// TwinCAT 3 PLC project PLC1_AssemblyLine
// Title: PLC1_AssemblyLine
// Company: Beckhoff Automation GmbH & Co. KG
// ProjectVersion: 1.0.0.0
// Description: Sample plc for the TcHmi_AssemblyLine training project
// ProgramVersion: 3.1.4020.10
// libraries:
//   Tc2_MC2, * (Beckhoff Automation GmbH)
//   Tc2_Standard, * (Beckhoff Automation GmbH)
//   Tc2_System, * (Beckhoff Automation GmbH)
//   Tc3_EventLogger, * (Beckhoff Automation GmbH)
//   Tc3_Module, * (Beckhoff Automation GmbH)
// project tree:
//   DUTs/ E_FeederAutoState.TcDUT, E_AxisMode.TcDUT, E_StationState.TcDUT, ST_HmiAxisInfo.TcDUT, ST_HmiFeederInfo.TcDUT, ST_Hmi.TcDUT, ST_HmiAutomaticMode.TcDUT, ST_HmiFeederRecipe.TcDUT, ST_HmiManualMode.TcDUT, ST_HmiOperationMode.TcDUT
//   GVLs/ GVL.TcGVL
//   / PlcTask.TcTTO
//   POUs/ deleteme.TcPOU, FB_Axis.TcPOU, FB_Feeder.TcPOU, MAIN.TcPOU
//   Project Information/ F_GetCompany.TcPOU, F_GetTitle.TcPOU, F_GetVersion.TcPOU
//   Version/ Global_Version.TcGVL
// real-time tasks:
//   TASK PlcTask: cycle T#10ms, priority 8, ADS port 350
// motion (NC):
//   TASK NC-Task-SAF: cycle T#2ms, priority 4, ADS port 501
//   TASK NC-Task-SVB: cycle T#10ms, priority 10, ADS port 511
//   AXIS Feeder1_AxisX (id 1)
//     OtherSettings: AllowMotionCmdToSlave=true
//     encoder EncType=1
//       SoftEndMinControl: Enable=true
//       SoftEndMaxControl: Enable=true, Range=1000
//     drive DrvType=5
//       TimeComp: TaskDelayCycles=1
//     controller CtrType=1
//       CtrPara: PriorControlFactor=1
//         Observer: BandWidth=20
//   AXIS Feeder1_AxisY (id 2)
//     OtherSettings: AllowMotionCmdToSlave=true
//     encoder EncType=1
//       SoftEndMinControl: Enable=true
//       SoftEndMaxControl: Enable=true, Range=1000
//     drive DrvType=5
//       TimeComp: TaskDelayCycles=1
//     controller CtrType=1
//       CtrPara: PriorControlFactor=1
//         Observer: BandWidth=20
//   AXIS Feeder2_AxisX (id 3)
//     OtherSettings: AllowMotionCmdToSlave=true
//     encoder EncType=1
//       SoftEndMinControl: Enable=true
//       SoftEndMaxControl: Enable=true, Range=1000
//     drive DrvType=5
//       TimeComp: TaskDelayCycles=1
//     controller CtrType=1
//       CtrPara: PriorControlFactor=1
//         Observer: BandWidth=20
//   AXIS Feeder2_AxisY (id 4)
//     OtherSettings: AllowMotionCmdToSlave=true
//     encoder EncType=1
//       SoftEndMinControl: Enable=true
//       SoftEndMaxControl: Enable=true, Range=1000
//     drive DrvType=5
//       TimeComp: TaskDelayCycles=1
//     controller CtrType=1
//       CtrPara: PriorControlFactor=1
//         Observer: BandWidth=20
// variable links:
//   PLC1_AssemblyLine/PLC1_AssemblyLine Instance <-> NC-Task-SAF/Axes/Feeder1_AxisX
//     PlcTask Inputs/MAIN.fbFeeders[1].fbAxisX.stAxis.NcToPlc <-> Outputs/ToPlc
//     PlcTask Outputs/MAIN.fbFeeders[1].fbAxisX.stAxis.PlcToNc <-> Inputs/FromPlc
//   PLC1_AssemblyLine/PLC1_AssemblyLine Instance <-> NC-Task-SAF/Axes/Feeder1_AxisY
//     PlcTask Inputs/MAIN.fbFeeders[1].fbAxisY.stAxis.NcToPlc <-> Outputs/ToPlc
//     PlcTask Outputs/MAIN.fbFeeders[1].fbAxisY.stAxis.PlcToNc <-> Inputs/FromPlc
//   PLC1_AssemblyLine/PLC1_AssemblyLine Instance <-> NC-Task-SAF/Axes/Feeder2_AxisX
//     PlcTask Inputs/MAIN.fbFeeders[2].fbAxisX.stAxis.NcToPlc <-> Outputs/ToPlc
//     PlcTask Outputs/MAIN.fbFeeders[2].fbAxisX.stAxis.PlcToNc <-> Inputs/FromPlc
//   PLC1_AssemblyLine/PLC1_AssemblyLine Instance <-> NC-Task-SAF/Axes/Feeder2_AxisY
//     PlcTask Inputs/MAIN.fbFeeders[2].fbAxisY.stAxis.NcToPlc <-> Outputs/ToPlc
//     PlcTask Outputs/MAIN.fbFeeders[2].fbAxisY.stAxis.PlcToNc <-> Inputs/FromPlc

CONFIGURATION PLC1_AssemblyLine
    RESOURCE PLC ON TwinCAT3
        TASK PlcTask(INTERVAL := T#10ms, PRIORITY := 8);
        PROGRAM MAIN WITH PlcTask : MAIN;
    END_RESOURCE
END_CONFIGURATION

// ---- DUTs/E_FeederAutoState.TcDUT
{attribute 'qualified_only'}
TYPE E_FeederAutoState :
(
	eState0_Reset				:= 0,
	eState1_MoveBackToTop		:= 1,
	eState2_MoveToTarget1PosX	:= 2,
	eState3_MoveToTarget1PosY	:= 3,
	eState4_Grab				:= 4,
	eState5_MoveBackToTop		:= 5,
	eState6_MoveToTarget2PosX	:= 6,
	eState7_MoveToTarget2PosY	:= 7,
	eState8_Place				:= 8
);
END_TYPE

// ---- DUTs/E_AxisMode.TcDUT
{attribute 'qualified_only'}
TYPE E_AxisMode :
(
	INIT,
	ENABLE,
	JOG,
	POSITIONING,
	STOP,
	RESET,
	ERROR
);
END_TYPE

// ---- DUTs/E_StationState.TcDUT
{attribute 'qualified_only'}
TYPE E_StationState :
(
	eAuto	:= 0,
	eManual := 1,
	eStop	:= 2	
);
END_TYPE

// ---- DUTs/ST_HmiAxisInfo.TcDUT
TYPE ST_HmiAxisInfo :
STRUCT
	//Actual position
	fActPosition	: LREAL;
	//Actual velocity
	fActVelocity	: LREAL;
	//Current state of axis
	nAxisState		: UDINT;
	//Current mode of axis
	eAxisMode		: E_AxisMode;
END_STRUCT
END_TYPE

// ---- DUTs/ST_HmiFeederInfo.TcDUT
TYPE ST_HmiFeederInfo :
STRUCT
	//Bundled information about axis X
	stAxisX				: ST_HmiAxisInfo;
	
	//Bundled information about axis Y
	stAxisY				: ST_HmiAxisInfo;
	
	//Information about the gripper
	bGripperIsClosed	: BOOL;
END_STRUCT
END_TYPE

// ---- DUTs/ST_Hmi.TcDUT
TYPE ST_Hmi :
STRUCT
	//Bundled operation mode settings and feedback
	stOperationMode			: ST_HmiOperationMode;		
	
	//Bundled manual mode settings and feedback
	stManualMode			: ST_HmiManualMode;
	
	//Bundled automatic mode settings and feedback
	stAutomaticMode			: ST_HmiAutomaticMode;
	
	//Bundled teach mode / recipe management settings and feedback
	stFeederRecipe			: ST_HmiFeederRecipe;
	
	//Bundled feeder information
	stFeederInfo			: ST_HmiFeederInfo;
END_STRUCT
END_TYPE

// ---- DUTs/ST_HmiAutomaticMode.TcDUT
TYPE ST_HmiAutomaticMode :
STRUCT
	//Current state of the automatic mode state machine
	nStateNumber		: E_FeederAutoState := 0;
	
	//Error simulation, state to in which should an error occure
	nErrorSimulation	: INT;
	
	fCurrentTargetPosX			: LREAL;
	fCurrentTargetPosY			: LREAL;
END_STRUCT
END_TYPE

// ---- DUTs/ST_HmiFeederRecipe.TcDUT
TYPE ST_HmiFeederRecipe :
STRUCT
	//Target 1 name
	sTarget1Name			: STRING := 'Target 1';
	//Target 1 positon for X axis
	fTarget1PositionX		: LREAL	:= LREAL#500.0;
	//Target 1 position for Y axis
	fTarget1PositionY		: LREAL	:= LREAL#500.0;

	//Target 2 name
	sTarget2Name			: STRING := 'Target 2';
	//Target 2 positon for X axis
	fTarget2PositionX		: LREAL	:= LREAL#1000.0;
	//Target 2 position for Y axis
	fTarget2PositionY		: LREAL	:= LREAL#1000.0;
	
	//Velocity of both axis	
	fVelocity				: LREAL := 50;
	
	//Recipe name
	sRecipeName				: STRING(50)	:= 'Default';
END_STRUCT
END_TYPE

// ---- DUTs/ST_HmiManualMode.TcDUT
TYPE ST_HmiManualMode :
STRUCT
	//Manual mode - move X axis forward
	bButtonForwardX			: BOOL;
	//Manual mode - move X axis backward
	bButtonBackwardX		: BOOL;
	//Manual mode - move Y axis forward
	bButtonForwardY		: BOOL;
	//Manual mode - move Y axis backward
	bButtonBackwardY		: BOOL;
	//Manual mode - close gripper
	bButtonCloseGripper		: BOOL;
	//Manual mode - velocity X axis in % of Reference Velocity	
	fVelocityX			: LREAL := 50;
	//Manual mode - velocity Y axis in % of Reference Velocity
	fVelocityY			: LREAL := 50;
END_STRUCT
END_TYPE

// ---- DUTs/ST_HmiOperationMode.TcDUT
TYPE ST_HmiOperationMode :
STRUCT
	//Set feeder into automatic mode
	bSetAutoMode		: BOOL;
	//Set feeder into manual mode
	bSetManualMode		: BOOL;
	//Set feeder into stop mode
	bSetStopMode		: BOOL;	
	
	
	//Feeder is in automatic mode
	bIsAutoMode			: BOOL;
	//Feeder is in manual mode
	bIsManualMode		: BOOL;
	//Feeder is in stop mode
	bIsStopMode			: BOOL;
	
END_STRUCT
END_TYPE

// ---- GVLs/GVL.TcGVL
{attribute 'qualified_only'}
VAR_GLOBAL
	bAxisError	: BOOL;
END_VAR

// ---- Version/Global_Version.TcGVL
{attribute 'TcGenerated'}
// This function has been automatically generated from the project information.
VAR_GLOBAL CONSTANT
	{attribute 'const_non_replaced'}
	{attribute 'linkalways'}
	stLibVersion_PLC1_AssemblyLine : ST_LibVersion := (iMajor := 1, iMinor := 0, iBuild := 0, iRevision := 0, sVersion := '1.0.0.0');
END_VAR

// ---- POUs/MAIN.TcPOU
PROGRAM MAIN
VAR
	//fbFeeder1		: FB_Feeder(nFeederId := 1);
	//fbFeeder2		: FB_Feeder(nFeederId := 2);
	
	fbFeeders		: ARRAY[1..2] OF FB_Feeder[(nFeederId := 1),(nFeederId := 2)];
END_VAR

//fbFeeder1();
//fbFeeder2();
fbFeeders[1]();
fbFeeders[2]();

END_PROGRAM

// ---- POUs/FB_Feeder.TcPOU
FUNCTION_BLOCK FB_Feeder
VAR_INPUT
END_VAR
VAR_OUTPUT
END_VAR
VAR
	//ID of the feeder as identification in hmi, log, etc.
	nFeederId					: USINT;

	//Current operation mode of the machine
	eStationState				: E_StationState;
	//Delay for simulating drag and drop
	fbTonAuto					: Tc2_Standard.TON;
	//State machine of automatic mode
	eAutoState					: E_FeederAutoState;
	fbAlarm						: Tc3_EventLogger.FB_TcAlarm;
	bWaitForErrorConfirmation	: BOOL;

	//NC-drive X axis
	fbAxisX						: FB_Axis;
	//NC-drive Y axis
	fbAxisY						: FB_Axis;	

	//Gripper status
	bCloseGripper				: BOOL;
	bGripperIsClosed			: BOOL;
	
	//Current position of the X axis for historize extension in the HMI server
	fHmiPosXHistorize			: LREAL;
	//Current position of the Y axis for historize extension in the HMI server
	fHmiPosYHistorize			: LREAL;
	//Current velocity of the X axis for historize extension in the HMI server
	fHmiVeloXHistorize			: LREAL;
	//Current velocity of the Y axis for historize extension in the HMI server
	fHmiVeloYHistorize			: LREAL;
	
	//Struct for communication with the HMI
	stHmi					: ST_Hmi;
END_VAR
VAR PERSISTENT
	//Current target positions from hmi recipe management
	stTargets				: ST_HmiFeederRecipe;
END_VAR

// Drives
fbAxisX();
fbAxisY();

// Hmi
M_Hmi();

// State machine
M_StationState();

// Events
M_Events();

IF stHmi.stOperationMode.bSetStopMode THEN
	IF eStationState = E_StationState.eStop THEN
		stHmi.stOperationMode.bSetStopMode := FALSE;
	END_IF
	eStationState := E_StationState.eStop;
ELSIF stHmi.stOperationMode.bSetAutoMode THEN
	IF eStationState = E_StationState.eAuto THEN
		stHmi.stOperationMode.bSetAutoMode := FALSE;
	END_IF
	eStationState := E_StationState.eAuto;
ELSIF stHmi.stOperationMode.bSetManualMode THEN
	IF eStationState = E_StationState.eManual THEN
		stHmi.stOperationMode.bSetManualMode := FALSE;
	END_IF
	eStationState := E_StationState.eManual;
END_IF

METHOD FB_init : BOOL
VAR_INPUT
	bInitRetains	: BOOL; // if TRUE, the retain variables are initialized (warm start / cold start)
	bInCopyCode		: BOOL;  // if TRUE, the instance afterwards gets moved into the copy code (online change)
	nFeederId		: USINT;
END_VAR
FeederId := nFeederId;
END_METHOD

PROPERTY PUBLIC FeederId : USINT
GET // PUBLIC
FeederId := THIS^.nFeederId;
END_GET
SET // PRIVATE
THIS^.nFeederId := FeederId;
END_SET
END_PROPERTY

METHOD PRIVATE M_Auto : HRESULT
VAR_INPUT
END_VAR
// Stoppping all axis for op mode change
IF stHmi.stOperationMode.bSetManualMode OR stHmi.stOperationMode.bSetStopMode THEN
	fbAxisX.bInStop := TRUE;
	fbAxisY.bInStop := TRUE;
	RETURN;
END_IF

fbTonAuto();
fbAxisX.fInOverride := LREAL#100;    
fbAxisX.fInVelocity := stTargets.fVelocity;
fbAxisY.fInOverride := LREAL#100;    
fbAxisY.fInVelocity := stTargets.fVelocity;

IF stHmi.stAutomaticMode.nErrorSimulation <> INT#0 AND NOT bWaitForErrorConfirmation AND_THEN eAutoState = stHmi.stAutomaticMode.nErrorSimulation THEN
	fbAlarm.CreateEx(TC_EVENTS.AssemblyLineEvents.AutomaticModeError, TRUE, 0);
	fbAlarm.ipArguments.Clear().AddInt(eAutoState);
	fbAlarm.Raise(0);
	bWaitForErrorConfirmation := TRUE;
END_IF

// State machine automatic mode
CASE eAutoState OF
	E_FeederAutoState.eState0_Reset:
		IF M_State0_Reset() = Tc3_Module.S_OK THEN
			IF M_CheckForError() = Tc3_Module.S_OK THEN
				eAutoState := E_FeederAutoState.eState1_MoveBackToTop;
			END_IF
		END_IF
	E_FeederAutoState.eState1_MoveBackToTop:
		IF M_State1_MoveBackToTop() = Tc3_Module.S_OK THEN
			IF M_CheckForError() = Tc3_Module.S_OK THEN
				eAutoState := E_FeederAutoState.eState2_MoveToTarget1PosX;
			END_IF
		END_IF
	E_FeederAutoState.eState2_MoveToTarget1PosX:
		IF M_State2_MoveToTarget1PosX() = Tc3_Module.S_OK THEN
			IF M_CheckForError() = Tc3_Module.S_OK THEN
				eAutoState := E_FeederAutoState.eState3_MoveToTarget1PosY;
			END_IF
		END_IF
	E_FeederAutoState.eState3_MoveToTarget1PosY:
		IF M_State3_MoveToTarget1PosY() = Tc3_Module.S_OK THEN
			IF M_CheckForError() = Tc3_Module.S_OK THEN
				eAutoState := E_FeederAutoState.eState4_Grab;
			END_IF
		END_IF
	E_FeederAutoState.eState4_Grab:
		IF M_State4_Grab() = Tc3_Module.S_OK THEN
			IF M_CheckForError() = Tc3_Module.S_OK THEN
				eAutoState := E_FeederAutoState.eState5_MoveBackToTop;
			END_IF
		END_IF
	E_FeederAutoState.eState5_MoveBackToTop:
		IF M_State5_MoveBackToTop() = Tc3_Module.S_OK THEN
			IF M_CheckForError() = Tc3_Module.S_OK THEN
				eAutoState := E_FeederAutoState.eState6_MoveToTarget2PosX;
			END_IF
		END_IF
	E_FeederAutoState.eState6_MoveToTarget2PosX:
		IF M_State6_MoveToTarget2PosX() = Tc3_Module.S_OK THEN
			IF M_CheckForError() = Tc3_Module.S_OK THEN
				eAutoState := E_FeederAutoState.eState7_MoveToTarget2PosY;
			END_IF
		END_IF
	E_FeederAutoState.eState7_MoveToTarget2PosY:
		IF M_State7_MoveToTarget2PosY() = Tc3_Module.S_OK THEN
			IF M_CheckForError() = Tc3_Module.S_OK THEN
				eAutoState := E_FeederAutoState.eState8_Place;
			END_IF
		END_IF
	E_FeederAutoState.eState8_Place:
		IF M_State8_Place() = Tc3_Module.S_OK THEN
			IF M_CheckForError() = Tc3_Module.S_OK THEN
				eAutoState := E_FeederAutoState.eState1_MoveBackToTop;
			END_IF
		END_IF
END_CASE
END_METHOD

METHOD PRIVATE M_CheckForError : HRESULT
VAR_INPUT
END_VAR
M_CheckForError := Tc3_Module.S_PENDING;
IF bWaitForErrorConfirmation THEN
	IF fbAlarm.eConfirmationState = TcEventConfirmationState.Confirmed THEN
		bWaitForErrorConfirmation := FALSE;
		stHmi.stAutomaticMode.nErrorSimulation := INT#0;
		fbAlarm.Clear(0, TRUE);
		M_CheckForError :=  Tc3_Module.S_OK;
	END_IF
ELSE
	M_CheckForError :=  Tc3_Module.S_OK;
END_IF
END_METHOD

METHOD PRIVATE M_Events : BOOL
VAR_INPUT
END_VAR
VAR
	sJsonAttributeAxis		: STRING;
END_VAR
VAR_INST
	fbTriggerAutomaticOn	: R_TRIG;
	fbTriggerManualModeOn	: R_TRIG;
	fbTriggerStop			: R_TRIG;
	fbTriggerErrorAxisX		: R_TRIG;
	fbTriggerErrorAxisY		: R_TRIG;	
	fbMessage 				: Tc3_EventLogger.FB_TcMessage;
	fbAlarmAxisX			: Tc3_EventLogger.FB_TcAlarm;
	fbAlarmAxisY			: Tc3_EventLogger.FB_TcAlarm;
END_VAR
fbTriggerAutomaticOn(CLK := eStationState = E_StationState.eAuto);
IF fbTriggerAutomaticOn.Q THEN
	fbMessage.CreateEx(TC_EVENTS.AssemblyLineEvents.FeederAutomaticOn, 0);
	fbMessage.ipArguments.Clear().AddUSInt(FeederId);
	fbMessage.Send(0);
END_IF

fbTriggerManualModeOn(CLK := eStationState = E_StationState.eManual);
IF fbTriggerManualModeOn.Q THEN
	fbMessage.CreateEx(TC_EVENTS.AssemblyLineEvents.FeederManualModeOn, 0);
	fbMessage.ipArguments.Clear().AddUSInt(FeederId);
	fbMessage.Send(0);
END_IF

fbTriggerStop(CLK := eStationState = E_StationState.eStop);
IF fbTriggerStop.Q THEN
	fbMessage.CreateEx(TC_EVENTS.AssemblyLineEvents.FeederStopped, 0);
	fbMessage.ipArguments.Clear().AddUSInt(FeederId);
	fbMessage.Send(0);
END_IF

fbTriggerErrorAxisX(CLK := fbAxisX.bOutError);
IF fbTriggerErrorAxisX.Q THEN
	fbAlarmAxisX.Clear(0, TRUE);
	fbAlarmAxisX.CreateEx(TC_EVENTS.AssemblyLineEvents.FeederError, FALSE, 0);
	fbAlarmAxisX.ipArguments.Clear().AddUSInt(FeederId).AddString('X');
	sJsonAttributeAxis := CONCAT(CONCAT('{"ErrorId: ', TO_STRING(fbAxisX.nOutErrorId)), '}');
	fbAlarmAxisX.SetJsonAttribute(sJsonAttributeAxis);
	fbAlarmAxisX.Raise(0);
END_IF

fbTriggerErrorAxisY(CLK := fbAxisY.bOutError);
IF fbTriggerErrorAxisY.Q THEN
	fbAlarmAxisY.Clear(0, TRUE);
	fbAlarmAxisY.CreateEx(TC_EVENTS.AssemblyLineEvents.FeederError, FALSE, 0);
	fbAlarmAxisY.ipArguments.Clear().AddUSInt(FeederId).AddString('Y');
	sJsonAttributeAxis := CONCAT(CONCAT('{"ErrorId: ', TO_STRING(fbAxisY.nOutErrorId)), '}');
	fbAlarmAxisY.SetJsonAttribute(sJsonAttributeAxis);
	fbAlarmAxisY.Raise(0);
END_IF
END_METHOD

METHOD M_Hmi : BOOL
VAR_INPUT
END_VAR
IF _TaskInfo[GETCURTASKINDEXEX()].FirstCycle THEN
	stHmi.stFeederRecipe := stTargets;
END_IF

stHmi.stOperationMode.bIsAutoMode := FALSE;
stHmi.stOperationMode.bIsManualMode := FALSE;
stHmi.stOperationMode.bIsStopMode := FALSE;
CASE eStationState OF
	E_StationState.eStop:
		stHmi.stOperationMode.bIsStopMode := TRUE;
	E_StationState.eAuto:
		stHmi.stOperationMode.bIsAutoMode := TRUE;
	E_StationState.eManual:
		stHmi.stOperationMode.bIsManualMode := TRUE;
END_CASE

stHmi.stAutomaticMode.nStateNumber := eAutoState;
stHmi.stFeederInfo.bGripperIsClosed := bGripperIsClosed;

// HMI historize actual position and velocity
fHmiPosXHistorize := fbAxisX.fOutActPosition;
fHmiPosYHistorize := fbAxisY.fOutActPosition;
fHmiVeloXHistorize := fbAxisX.fOutActVelocity;
fHmiVeloYHistorize := fbAxisY.fOutActVelocity;

// HMI axis information
stHmi.stFeederInfo.stAxisX.fActPosition := fbAxisX.fOutActPosition;
stHmi.stFeederInfo.stAxisX.fActVelocity := fbAxisX.fOutActVelocity;
stHmi.stFeederInfo.stAxisX.nAxisState := fbAxisX.nOutAxisState;
stHmi.stFeederInfo.stAxisX.eAxisMode := fbAxisX.eOutAxisMode;
stHmi.stAutomaticMode.fCurrentTargetPosX := fbAxisX.fInTargetPos;

stHmi.stFeederInfo.stAxisY.fActPosition := fbAxisY.fOutActPosition;
stHmi.stFeederInfo.stAxisY.fActVelocity := fbAxisY.fOutActVelocity;
stHmi.stFeederInfo.stAxisY.nAxisState := fbAxisY.nOutAxisState;
stHmi.stFeederInfo.stAxisY.eAxisMode := fbAxisY.eOutAxisMode;
stHmi.stAutomaticMode.fCurrentTargetPosY := fbAxisY.fInTargetPos;

//Set targets from hmi recipe management
stTargets := stHmi.stFeederRecipe;
END_METHOD

METHOD PRIVATE M_Manual : HRESULT
VAR_INPUT
END_VAR
// Stoppping all axis for op mode change
IF stHmi.stOperationMode.bSetAutoMode OR stHmi.stOperationMode.bSetStopMode THEN
	fbAxisX.bInStop := TRUE;
	fbAxisY.bInStop := TRUE;
	fbAxisX.bInJog := FALSE;
	fbAxisY.bInJog := FALSE;
	eAutoState := E_FeederAutoState.eState0_Reset;
	RETURN;
END_IF

fbAxisX.bInStop := FALSE;
fbAxisX.bInJog := TRUE;
fbAxisX.fInOverride := LREAL#100;
fbAxisX.fInVelocity := stHmi.stManualMode.fVelocityX;
fbAxisX.bInJogForward := stHmi.stManualMode.bButtonForwardX;
fbAxisX.bInJogBackward := stHmi.stManualMode.bButtonBackwardX;

fbAxisY.bInStop := FALSE;
fbAxisY.bInJog := TRUE;
fbAxisY.fInOverride := LREAL#100;
fbAxisY.fInVelocity := stHmi.stManualMode.fVelocityY;
fbAxisY.bInJogForward := stHmi.stManualMode.bButtonForwardY;
fbAxisY.bInJogBackward := stHmi.stManualMode.bButtonBackwardY;

bGripperIsClosed := bCloseGripper := stHmi.stManualMode.bButtonCloseGripper;
END_METHOD

METHOD PRIVATE M_State0_Reset : HRESULT
VAR_INPUT
END_VAR
M_State0_Reset := Tc3_Module.S_PENDING;
fbAxisX.fInTargetPos := 0.0;
fbAxisY.fInTargetPos := 0.0;
fbAxisX.bInStop := FALSE;
fbAxisY.bInStop := FALSE;

IF fbAxisX.fOutActPosition <> 0 THEN 
	fbAxisX.bInPositioning := TRUE;
END_IF

IF fbAxisY.fOutActPosition <> 0 THEN 
	fbAxisY.bInPositioning := TRUE;
END_IF

IF fbAxisX.fOutActPosition = 0 AND fbAxisY.fOutActPosition = 0 THEN 
	fbAxisX.bInPositioning := FALSE;
	fbAxisY.bInPositioning := FALSE;
	M_State0_Reset := Tc3_Module.S_OK;
END_IF
END_METHOD

METHOD PRIVATE M_State1_MoveBackToTop : HRESULT
VAR_INPUT
END_VAR
M_State1_MoveBackToTop :=  Tc3_Module.S_PENDING;
fbAxisY.fInTargetPos := 0.0;

IF fbAxisY.fOutActPosition <> 0 THEN
	fbAxisY.bInPositioning := TRUE;
ELSIF fbAxisY.fOutActPosition = 0 THEN 
	fbAxisY.bInPositioning := FALSE;
	M_State1_MoveBackToTop :=  Tc3_Module.S_OK;
END_IF
END_METHOD

METHOD PRIVATE M_State2_MoveToTarget1PosX : HRESULT
VAR_INPUT
END_VAR
M_State2_MoveToTarget1PosX := Tc3_Module.S_PENDING;
fbAxisX.fInTargetPos := stTargets.fTarget1PositionX;

IF fbAxisX.fOutActPosition <> stTargets.fTarget1PositionX THEN
	fbAxisX.bInPositioning := TRUE;
ELSIF fbAxisX.fOutActPosition = stTargets.fTarget1PositionX THEN 
	fbAxisX.bInPositioning := FALSE;
	M_State2_MoveToTarget1PosX := Tc3_Module.S_OK;
END_IF
END_METHOD

METHOD PRIVATE M_State3_MoveToTarget1PosY : HRESULT
VAR_INPUT
END_VAR
M_State3_MoveToTarget1PosY := Tc3_Module.S_PENDING;
fbAxisY.fInTargetPos := stTargets.fTarget1PositionY;

IF fbAxisY.fOutActPosition <> stTargets.fTarget1PositionY THEN
	fbAxisY.bInPositioning := TRUE;
ELSIF fbAxisY.fOutActPosition = stTargets.fTarget1PositionY THEN 
	fbAxisY.bInPositioning := FALSE;
	M_State3_MoveToTarget1PosY := Tc3_Module.S_OK;
END_IF
END_METHOD

METHOD PRIVATE M_State4_Grab : HRESULT
VAR_INPUT
END_VAR
M_State4_Grab := Tc3_Module.S_PENDING;
fbTonAuto.PT := T#2S;
fbTonAuto.IN := TRUE;
bCloseGripper := TRUE;

IF fbTonAuto.Q THEN
	fbTonAuto.IN := FALSE;
	bGripperIsClosed := TRUE;
	M_State4_Grab := Tc3_Module.S_OK;
END_IF
END_METHOD

METHOD PRIVATE M_State5_MoveBackToTop : HRESULT
VAR_INPUT
END_VAR
M_State5_MoveBackToTop := Tc3_Module.S_PENDING;
fbAxisY.fInTargetPos := 0.0;

IF fbAxisY.fOutActPosition <> 0 THEN
	fbAxisY.bInPositioning := TRUE;
ELSIF fbAxisY.fOutActPosition = 0 THEN 
	fbAxisY.bInPositioning := FALSE;
	M_State5_MoveBackToTop := Tc3_Module.S_OK;
END_IF
END_METHOD

METHOD PRIVATE M_State6_MoveToTarget2PosX : HRESULT
VAR_INPUT
END_VAR
M_State6_MoveToTarget2PosX := Tc3_Module.S_PENDING;
fbAxisX.fInTargetPos := stTargets.fTarget2PositionX;

IF fbAxisX.fOutActPosition <> stTargets.fTarget2PositionX THEN
	fbAxisX.bInPositioning := TRUE;
ELSIF fbAxisX.fOutActPosition = stTargets.fTarget2PositionX THEN 
	fbAxisX.bInPositioning := FALSE;
	M_State6_MoveToTarget2PosX := Tc3_Module.S_OK;
END_IF
END_METHOD

METHOD PRIVATE M_State7_MoveToTarget2PosY : HRESULT
VAR_INPUT
END_VAR
M_State7_MoveToTarget2PosY := Tc3_Module.S_PENDING;
fbAxisY.fInTargetPos := stTargets.fTarget2PositionY;

IF fbAxisY.fOutActPosition <> stTargets.fTarget2PositionY THEN
	fbAxisY.bInPositioning := TRUE;
ELSIF fbAxisY.fOutActPosition = stTargets.fTarget2PositionY THEN 
	fbAxisY.bInPositioning := FALSE;
	M_State7_MoveToTarget2PosY := Tc3_Module.S_OK;
END_IF
END_METHOD

METHOD PRIVATE M_State8_Place : HRESULT
VAR_INPUT
END_VAR
M_State8_Place := Tc3_Module.S_PENDING;
fbTonAuto.PT := T#2S;
fbTonAuto.IN := TRUE;
bCloseGripper := FALSE;

IF fbTonAuto.Q THEN
	fbTonAuto.IN := FALSE;
	bGripperIsClosed := FALSE;
	M_State8_Place := Tc3_Module.S_OK;
END_IF
END_METHOD

METHOD M_StationState : HRESULT
VAR_INPUT
END_VAR
VAR
END_VAR
CASE THIS^.eStationState OF
	E_StationState.eAuto:
		THIS^.M_Auto();
	E_StationState.eManual:
		THIS^.M_Manual();
	E_StationState.eStop:
		THIS^.M_Stop();	
END_CASE
END_METHOD

METHOD PRIVATE M_Stop : HRESULT
VAR_INPUT
END_VAR
fbAxisX.bInStop := TRUE;
fbAxisY.bInStop := TRUE;

IF stHmi.stOperationMode.bSetAutoMode THEN
	eAutoState := E_FeederAutoState.eState0_Reset;
END_IF
END_METHOD

END_FUNCTION_BLOCK

// ---- POUs/FB_Axis.TcPOU
FUNCTION_BLOCK FB_Axis
VAR_INPUT
	// Commands
	bInJog				: BOOL;
	bInJogForward		: BOOL;
	bInJogBackward		: BOOL;
	bInPositioning		: BOOL;
	bInStop				: BOOL;
	bInReset			: BOOL;

	// Parameters
	fInVelocity			: LREAL := 100.0;
	fInOverride			: LREAL := 100;
	fInTargetPos		: LREAL := 0;	
END_VAR
VAR_OUTPUT
	// Status
	bOutError			: BOOL;
	nOutErrorId			: UDINT;
	fOutActPosition		: DINT;
	fOutActVelocity		: DINT;
	fOutSetPosition		: LREAL;
	fOutSetVelocity		: LREAL;
	nOutAxisState		: UDINT;
	eOutAxisMode		: E_AxisMode;    
END_VAR
VAR
	// MC function blocks
	fbPower			: Tc2_MC2.MC_Power;
	fbReset			: Tc2_MC2.MC_Reset;
	fbStop			: Tc2_MC2.MC_Stop;	
	fbMoveAbs		: Tc2_MC2.MC_MoveAbsolute;
	fbJog			: Tc2_MC2.MC_Jog;
	
	// MC structures	
	stAxis			: Tc2_MC2.AXIS_REF;
	stPower			: Tc2_MC2.ST_McOutputs;
	stReset			: Tc2_MC2.ST_McOutputs;
	stStop			: Tc2_MC2.ST_McOutputs;
	stMoveAbs		: Tc2_MC2.ST_McOutputs;
	stJog			: Tc2_MC2.ST_McOutputs;
	
	// state machine
	eAxisMode		: E_AxisMode;
END_VAR
VAR CONSTANT
	fReferenceVelo	: LREAL:= 1000.00;
END_VAR

stAxis.ReadStatus();

// state machine
CASE eAxisMode OF

		E_AxisMode.INIT:
		
					fbPower.Enable := FALSE;
					fbReset.Execute := FALSE;
					fbStop.Execute := FALSE;
					fbMoveAbs.Execute := FALSE;
					fbJog.JogForward := FALSE;
					fbJog.JogBackwards := FALSE;
					eAxisMode := E_AxisMode.ENABLE;		
					
		E_AxisMode.ENABLE:					

					fbPower.Enable := TRUE;
					fbPower.Enable_Positive := TRUE;
					fbPower.Enable_Negative := TRUE;
					
					IF fbPower.Status THEN
						IF  bInStop THEN
							eAxisMode := E_AxisMode.STOP;						
						ELSIF  bInJog THEN
							eAxisMode := E_AxisMode.JOG;
						ELSIF bInPositioning THEN
							eAxisMode := E_AxisMode.POSITIONING;
						ELSIF  bInReset THEN
							eAxisMode := E_AxisMode.RESET;
						END_IF
					ELSIF fbPower.Error THEN
						eAxisMode := E_AxisMode.ERROR;						
					END_IF
					
					bOutError := fbPower.Error;
					nOutErrorId := fbPower.ErrorID;

		E_AxisMode.JOG: // Jog / manual mode with continuous speed *)					
        
					fbJog.Mode := Tc2_MC2.MC_JOGMODE_CONTINOUS;
					fbJog.Velocity := fReferenceVelo*fInVelocity/100.0;
					
					IF NOT bInStop THEN
						fbJog.JogForward := bInJogForward;
						fbJog.JogBackwards := bInJogBackward;					
					END_IF
					
					IF NOT bInJog THEN
						eAxisMode := E_AxisMode.STOP;
					END_IF 
					
					(* error state *)
					IF fbJog.Error THEN
						eAxisMode := E_AxisMode.ERROR;
					END_IF
					
					bOutError := fbJog.Error;
					nOutErrorId := fbJog.ErrorID;
		
		E_AxisMode.POSITIONING: // Positioning run
				
					IF bInPositioning AND NOT fbMoveAbs.Busy THEN
						fbMoveAbs.Velocity := fReferenceVelo*fInVelocity/100.00;
						fbMoveAbs.Position := fInTargetPos;
						fbMoveAbs.Execute := TRUE;
					END_IF
					
					// Wait for postioning run done
					IF fbMoveAbs.Done OR bInStop THEN
						bInPositioning := FALSE;
						fbMoveAbs.Execute := FALSE;
						eAxisMode := E_AxisMode.STOP;
					END_IF
					
					// Check if axis has an error
					IF fbMoveAbs.Error THEN
						eAxisMode := E_AxisMode.ERROR;
					END_IF
					
					bOutError := fbMoveAbs.Error;
					nOutErrorId := fbMoveAbs.ErrorID;	
					
		E_AxisMode.STOP: (* stops axis from continuos motion *)				
					fbStop.Execute := TRUE;
					IF fbStop.Active THEN
						fbStop.Execute := FALSE;
						bInStop := FALSE;
						IF fbStop.Done THEN
							bInStop := FALSE;
							eAxisMode := E_AxisMode.ENABLE;
						END_IF
					END_IF
					
					(* error state *)
					IF fbStop.Error THEN
						eAxisMode := E_AxisMode.ERROR;
					END_IF
					
					bOutError := fbStop.Error;
					nOutErrorId := fbStop.ErrorID;	

		E_AxisMode.RESET: //Reset drive to take new motion commands			

					fbReset.Execute := TRUE;
					IF fbReset.Busy THEN
						fbReset.Execute := FALSE;
						bInReset:= FALSE;
					END_IF
					IF fbReset.Done THEN
						eAxisMode := E_AxisMode.INIT;
					ELSIF fbReset.Error THEN
						eAxisMode := E_AxisMode.ERROR;
					END_IF
					
					bOutError := fbReset.Error;
					nOutErrorId := fbReset.ErrorID;

		E_AxisMode.ERROR:					

					IF stAxis.Status.Error THEN
						eAxisMode := E_AxisMode.RESET;
					ELSE
						eAxisMode := E_AxisMode.INIT;
					END_IF				

END_CASE

// Call MC function blocks
Power();
Reset();
Stop();
MoveAbs();
Jog();

// Status outputs
fOutActVelocity := TO_DINT(stAxis.NcToPlc.ActVelo);
fOutActPosition := TO_DINT(stAxis.NcToPlc.ActPos);
fOutSetVelocity := TO_LREAL(TO_DINT(stAxis.NcToPlc.SetVelo * 10000)) / 10000;
fOutSetPosition := TO_LREAL(TO_DINT(stAxis.NcToPlc.SetPos * 10000)) / 10000;
nOutAxisState := stAxis.NcToPlc.AxisState;
eOutAxisMode := eAxisMode;

ACTION Jog:
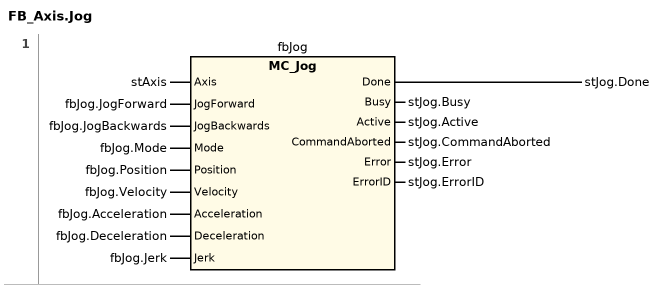
// NETWORK 1
fbJog(
    Axis := stAxis,
    JogForward := fbJog.JogForward,
    JogBackwards := fbJog.JogBackwards,
    Mode := fbJog.Mode,
    Position := fbJog.Position,
    Velocity := fbJog.Velocity,
    Acceleration := fbJog.Acceleration,
    Deceleration := fbJog.Deceleration,
    Jerk := fbJog.Jerk,
    Busy => stJog.Busy,
    Active => stJog.Active,
    CommandAborted => stJog.CommandAborted,
    Error => stJog.Error,
    ErrorID => stJog.ErrorID); // MC_Jog
stJog.Done := fbJog.Done;
END_ACTION

ACTION MoveAbs:
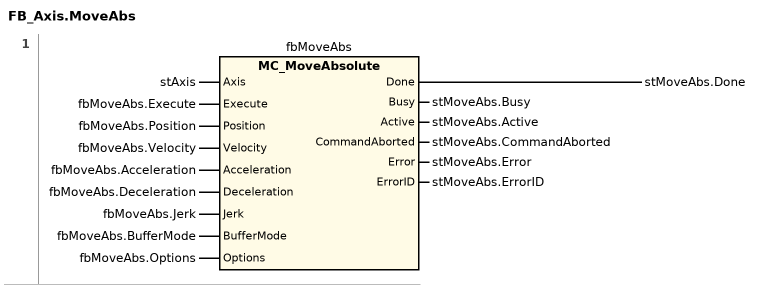
// NETWORK 1
fbMoveAbs(
    Axis := stAxis,
    Execute := fbMoveAbs.Execute,
    Position := fbMoveAbs.Position,
    Velocity := fbMoveAbs.Velocity,
    Acceleration := fbMoveAbs.Acceleration,
    Deceleration := fbMoveAbs.Deceleration,
    Jerk := fbMoveAbs.Jerk,
    BufferMode := fbMoveAbs.BufferMode,
    Options := fbMoveAbs.Options,
    Busy => stMoveAbs.Busy,
    Active => stMoveAbs.Active,
    CommandAborted => stMoveAbs.CommandAborted,
    Error => stMoveAbs.Error,
    ErrorID => stMoveAbs.ErrorID); // MC_MoveAbsolute
stMoveAbs.Done := fbMoveAbs.Done;
END_ACTION

ACTION Power:
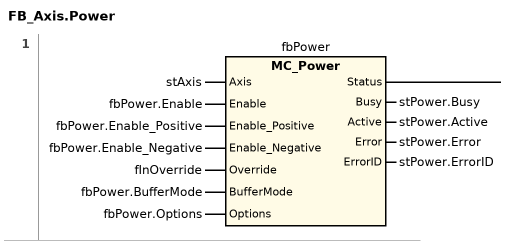
// NETWORK 1
fbPower(
    Axis := stAxis,
    Enable := fbPower.Enable,
    Enable_Positive := fbPower.Enable_Positive,
    Enable_Negative := fbPower.Enable_Negative,
    Override := fInOverride,
    BufferMode := fbPower.BufferMode,
    Options := fbPower.Options,
    Busy => stPower.Busy,
    Active => stPower.Active,
    Error => stPower.Error,
    ErrorID => stPower.ErrorID); // MC_Power
END_ACTION

ACTION Reset:
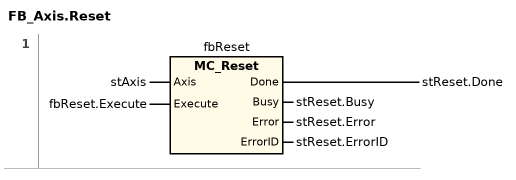
// NETWORK 1
fbReset(
    Axis := stAxis,
    Execute := fbReset.Execute,
    Busy => stReset.Busy,
    Error => stReset.Error,
    ErrorID => stReset.ErrorID); // MC_Reset
stReset.Done := fbReset.Done;
END_ACTION

ACTION Stop:
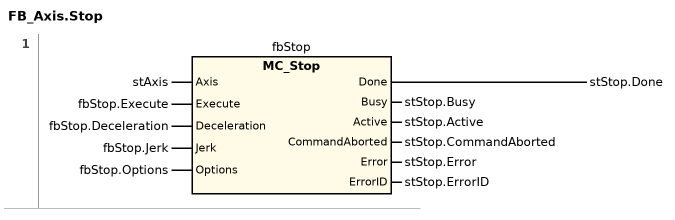
// NETWORK 1
fbStop(
    Axis := stAxis,
    Execute := fbStop.Execute,
    Deceleration := fbStop.Deceleration,
    Jerk := fbStop.Jerk,
    Options := fbStop.Options,
    Busy => stStop.Busy,
    Active => stStop.Active,
    CommandAborted => stStop.CommandAborted,
    Error => stStop.Error,
    ErrorID => stStop.ErrorID); // MC_Stop
stStop.Done := fbStop.Done;
END_ACTION

END_FUNCTION_BLOCK

// ---- POUs/deleteme.TcPOU
FUNCTION_BLOCK deleteme
VAR_INPUT
END_VAR
VAR_OUTPUT
END_VAR
VAR
END_VAR

END_FUNCTION_BLOCK

// ---- Project Information/F_GetCompany.TcPOU
// This function has been automatically generated from the project information.
{attribute 'signature_flag' := '1073741824'}
{attribute 'TcGenerated'}
{attribute 'no-analysis'}
FUNCTION F_GetCompany : WSTRING
VAR_INPUT
	
END_VAR

F_GetCompany := "Beckhoff Automation GmbH & Co. KG";

END_FUNCTION

// ---- Project Information/F_GetTitle.TcPOU
// This function has been automatically generated from the project information.
{attribute 'signature_flag' := '1073741824'}
{attribute 'TcGenerated'}
{attribute 'no-analysis'}
FUNCTION F_GetTitle : WSTRING
VAR_INPUT
	
END_VAR

F_GetTitle := "PLC1_AssemblyLine";

END_FUNCTION

// ---- Project Information/F_GetVersion.TcPOU
// This function has been automatically generated from the project information.
{attribute 'signature_flag' := '1073741824'}
{attribute 'TcGenerated'}
{attribute 'no-analysis'}
FUNCTION F_GetVersion : ST_LibVersion
VAR_INPUT
	
END_VAR

F_GetVersion.iMajor := 1;
F_GetVersion.iMinor := 0;
F_GetVersion.iBuild := 0;
F_GetVersion.iRevision := 0;

END_FUNCTION
